GLOBALCONSTANTS AID_GC (* Graphic context object attribute ids *)
  (* Standard: 61499-1; Description: Copyright (c) 2023 HR Agrartechnik GmbH This program and the accompanying materials are made available under the terms of the Eclipse Public License 2.0 which is available at https://www.eclipse.org/legal/epl-2.0/ SPDX-License-Identifier: EPL-2.0 *)
  (* Version 1.0, 2026-06-20, Franz Höpfinger, HR Agrartechnik GmbH *)
  PACKAGE isobus::UT::Q::const::AID;
  VAR_GLOBAL CONSTANT
    VP_WIDTH : USINT := USINT#1; (* 1: AID_GC_VP_WIDTH *)
    VP_HEIGHT : USINT := USINT#2; (* 2: AID_GC_VP_HEIGHT *)
    VP_X : USINT := USINT#3; (* 3: AID_GC_VP_X *)
    VP_Y : USINT := USINT#4; (* 4: AID_GC_VP_Y *)
    CANVAS_WIDTH : USINT := USINT#5; (* 5: AID_GC_CANVAS_WIDTH *)
    CANVAS_HEIGHT : USINT := USINT#6; (* 6: AID_GC_CANVAS_HEIGHT *)
    VP_ZOOM : USINT := USINT#7; (* 7: AID_GC_VP_ZOOM *)
    GR_CURSOR_X : USINT := USINT#8; (* 8: AID_GC_GR_CURSOR_X *)
    GR_CURSOR_Y : USINT := USINT#9; (* 9: AID_GC_GR_CURSOR_Y *)
    FG_COLOUR : USINT := USINT#10; (* 10: AID_GC_FG_COLOUR *)
    BACKGROUND_COLOUR : USINT := USINT#11; (* 11: AID_GC_BACKGROUND_COLOUR - Background colour index. *)
    FONT_ATT : USINT := USINT#12; (* 12: AID_GC_FONT_ATT - Object ID of a Font Attributes object. *)
    LINE_ATT : USINT := USINT#13; (* 13: AID_GC_LINE_ATT - Object ID of a Line Attributes object. *)
    FILL_ATT : USINT := USINT#14; (* 14: AID_GC_FILL_ATT - Object ID of a Fill Attributes object. *)
    FORMAT : USINT := USINT#15; (* 15: AID_GC_FORMAT - Canvas Type: 0 = Monochrome, 1 = 4-bit colour, 2 = 8-bit colour. *)
    OPTIONS : USINT := USINT#16; (* 16: AID_GC_OPTIONS - Bitmask: Bit 0=Transparency (0=opaque, 1=transparent), Bit 1=Colour mode *)
    TRANS_COLOUR : USINT := USINT#17; (* 17: AID_GC_TRANS_COLOUR *)
  END_VAR
END_GLOBALCONSTANTS
